TYPE ST_PLCPersistentVars :
STRUCT
	Hardsettings					: ST_HardSettings; 
	Softsettings					: ST_Softsettings;
END_STRUCT
END_TYPE

(* stored: Version 1.1.0.1, ProductVersion 3.1.4026.18
   DUT ST_PLCPersistentVars: Id {3c1dacfe-1e38-45b6-bfef-fee6afbebfcc} *)
